// TIA Portal V19 export
TYPE "LAF_typeXXXProductionParameters"
// stored: Access Published
   STRUCT
      upperVel : LReal := 100.0;   // 产品模式速度上限
      vel : LReal := 20.0;   // 产品模式设定值，画面做限制根据上限值如果超了不允许输入
      distanceList : Array[0..99] of "LBC_typeAxis16PosSetPosition";
      acc : LReal := 0.5;
      dec : LReal := 0.5;
   END_STRUCT;
END_TYPE
